(* IEC 61131-3 sources: Industry-PLC-LLM/data/PLCBEAD_repo/PLCBEAD_PLCEmbed-main/PLC-BEAD/Source/GEB/WORD_OF_BYTE, 1 file *)

(* ---- WORD_OF_BYTE.ST ---- *)
FUNCTION WORD_OF_BYTE:WORD
	VAR_INPUT
		B1 :	BYTE;
		B0 :	BYTE;
	END_VAR
	WORD_OF_BYTE := SHL(BYTE_TO_WORD(B1),8) OR BYTE_TO_WORD(B0);
END_FUNCTION

PROGRAM program0
  	VAR
		B1 :	BYTE;
		B0 :	BYTE;
		CEIL5_OUT : WORD;
	END_VAR

  	CEIL5_OUT := WORD_OF_BYTE(B1, B0);
END_PROGRAM
